INTERFACE ITF_Group3 EXTENDS ITF_BaseGroupElement

END_INTERFACE

(* stored: Version 1.1.0.1
   Itf ITF_Group3: Id {d2772093-7c02-0780-0cee-c4aaffeeb2ce} *)
